TYPE ST_TcMatSimObjectDataAreaInfo :
STRUCT
	pPlcVar: PVOID;
	pModuleProcImg: PVOID;
	nSize: UDINT;
	nDataAreaId: UDINT;
	eDataAreaType: E_TcMatSimDataAreaType;
END_STRUCT
END_TYPE

(* stored: Version 1.1.0.1, ProductVersion 3.1.4024.4
   DUT ST_TcMatSimObjectDataAreaInfo: Id {b5bb7ee5-267f-4be5-9aea-789179337215} *)
